FUNCTION_BLOCK FB_Square IMPLEMENTS I_Shape


METHOD M_Draw : BOOL
ADSLOGSTR(ADSLOG_MSGTYPE_HINT, 'Draw Square', '');
M_Draw := TRUE;
END_METHOD

END_FUNCTION_BLOCK

(* stored: Version 1.1.0.1, ProductVersion 3.1.4024.12
   POU FB_Square: Id {6850b2a4-8187-4978-aaec-3d3752789de4}, SpecialFunc None
   Method M_Draw: Id {e315df57-dcd2-4e04-a747-7cbc334673e3} *)
